DATA_BLOCK "Tor2_RecepturyStacjaMycia"   // DB6
VERSION : 0.1
// stored: AutoNumber true, DBAccessibleFromOPCUA true, InstanceOfName FB_RecepturyStacjaMycia, InstanceOfType FB
"FB_RecepturyStacjaMycia"
BEGIN
   Receptura[0].nazwaReceptury := WSTRING#'Technology';
   Receptura[1].nazwaReceptury := WSTRING#'CIP AGENTS';
   Receptura[2].nazwaReceptury := WSTRING#'CIP Internal';
   Receptura[3].nazwaReceptury := WSTRING#'Technology';
   Receptura[4].nazwaReceptury := WSTRING#'Pasteurizer line';
   Receptura[5].nazwaReceptury := WSTRING#'NF line';
   Receptura[6].nazwaReceptury := WSTRING#'Car line';
   Receptura[7].nazwaReceptury := WSTRING#'Cream line';
   Receptura[8].nazwaReceptury := WSTRING#'Cream line [test]';
   Receptura[9..19].nazwaReceptury := WSTRING#'nazwa receptury';
   Receptura[20].nazwaReceptury := WSTRING#'Cream line';
   Receptura[0].Krok[0..1].nazwaKroku := WSTRING#'Płukanie Zimne';
   Receptura[0].Krok[2].nazwaKroku := WSTRING#'Płukanie Gorące';
   Receptura[0].Krok[3].nazwaKroku := WSTRING#'Ług';
   Receptura[0].Krok[4].nazwaKroku := WSTRING#'Kwas';
   Receptura[0].Krok[5].nazwaKroku := WSTRING#'Płukanie Główne';
   Receptura[0].Krok[6].nazwaKroku := WSTRING#'Dezynfekcja';
   Receptura[1].Krok[0].nazwaKroku := WSTRING#'Płukanie Zimne';
   Receptura[1].Krok[1].nazwaKroku := WSTRING#'Холодне полоскание';
   Receptura[1].Krok[2].nazwaKroku := WSTRING#'Горячее полоскание';
   Receptura[1].Krok[3].nazwaKroku := WSTRING#'ЩЕЛОЧЬ';
   Receptura[1].Krok[4].nazwaKroku := WSTRING#'КИСЛОТА';
   Receptura[1].Krok[5].nazwaKroku := WSTRING#'полоскание';
   Receptura[1].Krok[6].nazwaKroku := WSTRING#'Дезинфекция';
   Receptura[2].Krok[0].nazwaKroku := WSTRING#'Plukanie zimne';
   Receptura[2].Krok[1].nazwaKroku := WSTRING#'Холодне полоскание';
   Receptura[2].Krok[2].nazwaKroku := WSTRING#'Горячее полоскание';
   Receptura[2].Krok[3].nazwaKroku := WSTRING#'ЩЕЛОЧЬ';
   Receptura[2].Krok[4].nazwaKroku := WSTRING#'КИСЛОТА';
   Receptura[2].Krok[5].nazwaKroku := WSTRING#'полоскание';
   Receptura[2].Krok[6].nazwaKroku := WSTRING#'CIP Agents';
   Receptura[3].Krok[0].nazwaKroku := WSTRING#'Płukanie Główne';
   Receptura[3].Krok[1].nazwaKroku := WSTRING#'Холодне полоскание';
   Receptura[3].Krok[2].nazwaKroku := WSTRING#'Горячее полоскание';
   Receptura[3].Krok[3].nazwaKroku := WSTRING#'ЩЕЛОЧЬ';
   Receptura[3].Krok[4].nazwaKroku := WSTRING#'КИСЛОТА';
   Receptura[3].Krok[5].nazwaKroku := WSTRING#'полоскание';
   Receptura[3].Krok[6].nazwaKroku := WSTRING#'Dezynfekcja';
   Receptura[4].Krok[0].nazwaKroku := WSTRING#'Ług';
   Receptura[4].Krok[1].nazwaKroku := WSTRING#'Холодне полоскание';
   Receptura[4].Krok[2].nazwaKroku := WSTRING#'Горячее полоскание';
   Receptura[4].Krok[3].nazwaKroku := WSTRING#'ЩЕЛОЧЬ';
   Receptura[4].Krok[4].nazwaKroku := WSTRING#'КИСЛОТА';
   Receptura[4].Krok[5].nazwaKroku := WSTRING#'полоскание';
   Receptura[4].Krok[6].nazwaKroku := WSTRING#'Dezynfekcja';
   Receptura[5].Krok[0].nazwaKroku := WSTRING#'Kwas';
   Receptura[5].Krok[1].nazwaKroku := WSTRING#'Холодне полоскание';
   Receptura[5].Krok[2].nazwaKroku := WSTRING#'Горячее полоскание';
   Receptura[5].Krok[3].nazwaKroku := WSTRING#'ЩЕЛОЧЬ';
   Receptura[5].Krok[4].nazwaKroku := WSTRING#'КИСЛОТА';
   Receptura[5].Krok[5].nazwaKroku := WSTRING#'полоскание';
   Receptura[5].Krok[6].nazwaKroku := WSTRING#'Dezynfekcja';
   Receptura[6].Krok[0].nazwaKroku := WSTRING#'Ług';
   Receptura[6].Krok[1].nazwaKroku := WSTRING#'Холодне полоскание';
   Receptura[6].Krok[2].nazwaKroku := WSTRING#'Горячее полоскание';
   Receptura[6].Krok[3].nazwaKroku := WSTRING#'ЩЕЛОЧЬ';
   Receptura[6].Krok[4].nazwaKroku := WSTRING#'КИСЛОТА';
   Receptura[6].Krok[5].nazwaKroku := WSTRING#'полоскание';
   Receptura[6].Krok[6].nazwaKroku := WSTRING#'Dezynfekcja';
   Receptura[7].Krok[0].nazwaKroku := WSTRING#'Płukanie Główne';
   Receptura[7].Krok[1].nazwaKroku := WSTRING#'Холодне полоскание';
   Receptura[7].Krok[2].nazwaKroku := WSTRING#'Горячее полоскание';
   Receptura[7].Krok[3].nazwaKroku := WSTRING#'ЩЕЛОЧЬ';
   Receptura[7].Krok[4].nazwaKroku := WSTRING#'КИСЛОТА';
   Receptura[7].Krok[5].nazwaKroku := WSTRING#'полоскание';
   Receptura[7].Krok[6].nazwaKroku := WSTRING#'Dezynfekcja';
   Receptura[8].Krok[0].nazwaKroku := WSTRING#'Płukanie Gorące';
   Receptura[8].Krok[1].nazwaKroku := WSTRING#'Холодне полоскание';
   Receptura[8].Krok[2].nazwaKroku := WSTRING#'Горячее полоскание';
   Receptura[8].Krok[3].nazwaKroku := WSTRING#'ЩЕЛОЧЬ';
   Receptura[8].Krok[4].nazwaKroku := WSTRING#'КИСЛОТА';
   Receptura[8].Krok[5].nazwaKroku := WSTRING#'Płukanie Główne';
   Receptura[8].Krok[6].nazwaKroku := WSTRING#'Dezynfekcja';
   Receptura[9].Krok[0].nazwaKroku := WSTRING#'';
   Receptura[9].Krok[1].nazwaKroku := WSTRING#'Płukanie Zimne';
   Receptura[9].Krok[2].nazwaKroku := WSTRING#'Płukanie Gorące';
   Receptura[9].Krok[3].nazwaKroku := WSTRING#'Ług';
   Receptura[9].Krok[4].nazwaKroku := WSTRING#'Kwas';
   Receptura[9].Krok[5].nazwaKroku := WSTRING#'Płukanie Główne';
   Receptura[9].Krok[6].nazwaKroku := WSTRING#'Dezynfekcja';
   Receptura[10].Krok[0].nazwaKroku := WSTRING#'';
   Receptura[10].Krok[1].nazwaKroku := WSTRING#'Płukanie Zimne';
   Receptura[10].Krok[2].nazwaKroku := WSTRING#'Płukanie Gorące';
   Receptura[10].Krok[3].nazwaKroku := WSTRING#'Ług';
   Receptura[10].Krok[4].nazwaKroku := WSTRING#'Kwas';
   Receptura[10].Krok[5].nazwaKroku := WSTRING#'Płukanie Główne';
   Receptura[10].Krok[6].nazwaKroku := WSTRING#'Dezynfekcja';
   Receptura[11].Krok[0].nazwaKroku := WSTRING#'';
   Receptura[11].Krok[1].nazwaKroku := WSTRING#'Płukanie Zimne';
   Receptura[11].Krok[2].nazwaKroku := WSTRING#'Płukanie Gorące';
   Receptura[11].Krok[3].nazwaKroku := WSTRING#'Ług';
   Receptura[11].Krok[4].nazwaKroku := WSTRING#'Kwas';
   Receptura[11].Krok[5].nazwaKroku := WSTRING#'Płukanie Główne';
   Receptura[11].Krok[6].nazwaKroku := WSTRING#'Dezynfekcja';
   Receptura[12].Krok[0].nazwaKroku := WSTRING#'';
   Receptura[12].Krok[1].nazwaKroku := WSTRING#'Płukanie Zimne';
   Receptura[12].Krok[2].nazwaKroku := WSTRING#'Płukanie Gorące';
   Receptura[12].Krok[3].nazwaKroku := WSTRING#'Ług';
   Receptura[12].Krok[4].nazwaKroku := WSTRING#'Kwas';
   Receptura[12].Krok[5].nazwaKroku := WSTRING#'Płukanie Główne';
   Receptura[12].Krok[6].nazwaKroku := WSTRING#'Dezynfekcja';
   Receptura[13].Krok[0].nazwaKroku := WSTRING#'';
   Receptura[13].Krok[1].nazwaKroku := WSTRING#'Płukanie Zimne';
   Receptura[13].Krok[2].nazwaKroku := WSTRING#'Płukanie Gorące';
   Receptura[13].Krok[3].nazwaKroku := WSTRING#'Ług';
   Receptura[13].Krok[4].nazwaKroku := WSTRING#'Kwas';
   Receptura[13].Krok[5].nazwaKroku := WSTRING#'Płukanie Główne';
   Receptura[13].Krok[6].nazwaKroku := WSTRING#'Dezynfekcja';
   Receptura[14].Krok[0].nazwaKroku := WSTRING#'';
   Receptura[14].Krok[1].nazwaKroku := WSTRING#'Płukanie Zimne';
   Receptura[14].Krok[2].nazwaKroku := WSTRING#'Płukanie Gorące';
   Receptura[14].Krok[3].nazwaKroku := WSTRING#'Ług';
   Receptura[14].Krok[4].nazwaKroku := WSTRING#'Kwas';
   Receptura[14].Krok[5].nazwaKroku := WSTRING#'Płukanie Główne';
   Receptura[14].Krok[6].nazwaKroku := WSTRING#'Dezynfekcja';
   Receptura[15].Krok[0].nazwaKroku := WSTRING#'';
   Receptura[15].Krok[1].nazwaKroku := WSTRING#'Płukanie Zimne';
   Receptura[15].Krok[2].nazwaKroku := WSTRING#'Płukanie Gorące';
   Receptura[15].Krok[3].nazwaKroku := WSTRING#'Ług';
   Receptura[15].Krok[4].nazwaKroku := WSTRING#'Kwas';
   Receptura[15].Krok[5].nazwaKroku := WSTRING#'Płukanie Główne';
   Receptura[15].Krok[6].nazwaKroku := WSTRING#'Dezynfekcja';
   Receptura[16].Krok[0].nazwaKroku := WSTRING#'';
   Receptura[16].Krok[1].nazwaKroku := WSTRING#'Płukanie Zimne';
   Receptura[16].Krok[2].nazwaKroku := WSTRING#'Płukanie Gorące';
   Receptura[16].Krok[3].nazwaKroku := WSTRING#'Ług';
   Receptura[16].Krok[4].nazwaKroku := WSTRING#'Kwas';
   Receptura[16].Krok[5].nazwaKroku := WSTRING#'Płukanie Główne';
   Receptura[16].Krok[6].nazwaKroku := WSTRING#'Dezynfekcja';
   Receptura[17].Krok[0].nazwaKroku := WSTRING#'';
   Receptura[17].Krok[1].nazwaKroku := WSTRING#'Płukanie Zimne';
   Receptura[17].Krok[2].nazwaKroku := WSTRING#'Płukanie Gorące';
   Receptura[17].Krok[3].nazwaKroku := WSTRING#'Ług';
   Receptura[17].Krok[4].nazwaKroku := WSTRING#'Kwas';
   Receptura[17].Krok[5].nazwaKroku := WSTRING#'Płukanie Główne';
   Receptura[17].Krok[6].nazwaKroku := WSTRING#'Dezynfekcja';
   Receptura[18].Krok[0].nazwaKroku := WSTRING#'';
   Receptura[18].Krok[1].nazwaKroku := WSTRING#'Płukanie Zimne';
   Receptura[18].Krok[2].nazwaKroku := WSTRING#'Płukanie Gorące';
   Receptura[18].Krok[3].nazwaKroku := WSTRING#'Ług';
   Receptura[18].Krok[4].nazwaKroku := WSTRING#'Kwas';
   Receptura[18].Krok[5].nazwaKroku := WSTRING#'Płukanie Główne';
   Receptura[18].Krok[6].nazwaKroku := WSTRING#'Dezynfekcja';
   Receptura[19].Krok[0].nazwaKroku := WSTRING#'';
   Receptura[19].Krok[1].nazwaKroku := WSTRING#'Płukanie Zimne';
   Receptura[19].Krok[2].nazwaKroku := WSTRING#'Płukanie Gorące';
   Receptura[19].Krok[3].nazwaKroku := WSTRING#'Ług';
   Receptura[19].Krok[4].nazwaKroku := WSTRING#'Kwas';
   Receptura[19].Krok[5].nazwaKroku := WSTRING#'Płukanie Główne';
   Receptura[19].Krok[6].nazwaKroku := WSTRING#'Dezynfekcja';
   Receptura[20].Krok[0..1].nazwaKroku := WSTRING#'Płukanie Zimne';
   Receptura[20].Krok[2].nazwaKroku := WSTRING#'Płukanie Gorące';
   Receptura[20].Krok[3].nazwaKroku := WSTRING#'Ług';
   Receptura[20].Krok[4].nazwaKroku := WSTRING#'Kwas';
   Receptura[20].Krok[5].nazwaKroku := WSTRING#'Płukanie Główne';
   Receptura[20].Krok[6].nazwaKroku := WSTRING#'Dezynfekcja';
   Receptura[0].Krok[0].PM[0] := 0.0;
   Receptura[0].Krok[0].PM[1] := 1.0;
   Receptura[0].Krok[0].PM[2] := 20.0;
   Receptura[0].Krok[0].PM[3] := 10.0;
   Receptura[0].Krok[0].PM[4] := 120.0;
   Receptura[0].Krok[0].PM[5] := 1.0;
   Receptura[0].Krok[0].PM[6..11] := 0.0;
   Receptura[0].Krok[0].PM[12] := 3.0;
   Receptura[0].Krok[0].PM[13..14] := 0.0;
   Receptura[0].Krok[0].PM[15] := 1.0;
   Receptura[0].Krok[0].PM[16..18] := 0.0;
   Receptura[0].Krok[0].PM[19] := 300.0;
   Receptura[0].Krok[0].PM[20] := 0.0;
   Receptura[0].Krok[0].PM[21] := 1.0;
   Receptura[0].Krok[0].PM[22..23] := 0.0;
   Receptura[0].Krok[0].PM[24] := 2102.0;
   Receptura[0].Krok[0].PM[25..30] := 0.0;
   Receptura[0].Krok[1].PM[0] := 0.0;
   Receptura[0].Krok[1].PM[1] := 1.0;
   Receptura[0].Krok[1].PM[2] := 20.0;
   Receptura[0].Krok[1].PM[3] := 10.0;
   Receptura[0].Krok[1].PM[4] := 120.0;
   Receptura[0].Krok[1].PM[5] := 1.0;
   Receptura[0].Krok[1].PM[6..11] := 0.0;
   Receptura[0].Krok[1].PM[12] := 3.0;
   Receptura[0].Krok[1].PM[13..14] := 0.0;
   Receptura[0].Krok[1].PM[15] := 1.0;
   Receptura[0].Krok[1].PM[16..18] := 0.0;
   Receptura[0].Krok[1].PM[19] := 300.0;
   Receptura[0].Krok[1].PM[20] := 0.0;
   Receptura[0].Krok[1].PM[21] := 1.0;
   Receptura[0].Krok[1].PM[22..23] := 0.0;
   Receptura[0].Krok[1].PM[24] := 2102.0;
   Receptura[0].Krok[1].PM[25..30] := 0.0;
   Receptura[0].Krok[2].PM[0] := 0.0;
   Receptura[0].Krok[2].PM[1] := 1.0;
   Receptura[0].Krok[2].PM[2] := 20.0;
   Receptura[0].Krok[2].PM[3] := 10.0;
   Receptura[0].Krok[2].PM[4] := 120.0;
   Receptura[0].Krok[2].PM[5] := 0.5;
   Receptura[0].Krok[2].PM[6..11] := 0.0;
   Receptura[0].Krok[2].PM[12] := 3.0;
   Receptura[0].Krok[2].PM[13] := 0.0;
   Receptura[0].Krok[2].PM[14] := 30.0;
   Receptura[0].Krok[2].PM[15] := 1.0;
   Receptura[0].Krok[2].PM[16] := 10.0;
   Receptura[0].Krok[2].PM[17..18] := 0.0;
   Receptura[0].Krok[2].PM[19] := 300.0;
   Receptura[0].Krok[2].PM[20] := 0.0;
   Receptura[0].Krok[2].PM[21] := 1.0;
   Receptura[0].Krok[2].PM[22..23] := 0.0;
   Receptura[0].Krok[2].PM[24] := 2102.0;
   Receptura[0].Krok[2].PM[25..30] := 0.0;
   Receptura[0].Krok[3].PM[0] := 0.0;
   Receptura[0].Krok[3].PM[1] := 1.0;
   Receptura[0].Krok[3].PM[2] := 20.0;
   Receptura[0].Krok[3].PM[3] := 10.0;
   Receptura[0].Krok[3].PM[4] := 120.0;
   Receptura[0].Krok[3].PM[5] := 1.0;
   Receptura[0].Krok[3].PM[6] := 900.0;
   Receptura[0].Krok[3].PM[7..9] := 0.0;
   Receptura[0].Krok[3].PM[10] := 40.0;
   Receptura[0].Krok[3].PM[11] := 75.0;
   Receptura[0].Krok[3].PM[12] := 3.0;
   Receptura[0].Krok[3].PM[13] := 70.0;
   Receptura[0].Krok[3].PM[14] := 30.0;
   Receptura[0].Krok[3].PM[15] := 1.0;
   Receptura[0].Krok[3].PM[16] := 10.0;
   Receptura[0].Krok[3].PM[17] := 2.05;
   Receptura[0].Krok[3].PM[18] := 20.0;
   Receptura[0].Krok[3].PM[19] := 300.0;
   Receptura[0].Krok[3].PM[20] := 0.0;
   Receptura[0].Krok[3].PM[21..22] := 1.0;
   Receptura[0].Krok[3].PM[23] := 0.0;
   Receptura[0].Krok[3].PM[24] := 2102.0;
   Receptura[0].Krok[3].PM[25..30] := 0.0;
   Receptura[0].Krok[4].PM[0] := 0.0;
   Receptura[0].Krok[4].PM[1] := 1.0;
   Receptura[0].Krok[4].PM[2] := 20.0;
   Receptura[0].Krok[4].PM[3] := 10.0;
   Receptura[0].Krok[4].PM[4] := 120.0;
   Receptura[0].Krok[4].PM[5] := 0.1;
   Receptura[0].Krok[4].PM[6] := 300.0;
   Receptura[0].Krok[4].PM[7..9] := 0.0;
   Receptura[0].Krok[4].PM[10] := 30.0;
   Receptura[0].Krok[4].PM[11] := 50.0;
   Receptura[0].Krok[4].PM[12] := 3.0;
   Receptura[0].Krok[4].PM[13] := 55.0;
   Receptura[0].Krok[4].PM[14] := 0.0;
   Receptura[0].Krok[4].PM[15] := 1.0;
   Receptura[0].Krok[4].PM[16] := 10.0;
   Receptura[0].Krok[4].PM[17] := 1.75;
   Receptura[0].Krok[4].PM[18] := 20.0;
   Receptura[0].Krok[4].PM[19] := 300.0;
   Receptura[0].Krok[4].PM[20] := 0.0;
   Receptura[0].Krok[4].PM[21..22] := 1.0;
   Receptura[0].Krok[4].PM[23] := 0.0;
   Receptura[0].Krok[4].PM[24] := 2102.0;
   Receptura[0].Krok[4].PM[25..30] := 0.0;
   Receptura[0].Krok[5].PM[0] := 0.0;
   Receptura[0].Krok[5].PM[1] := 1.0;
   Receptura[0].Krok[5].PM[2] := 20.0;
   Receptura[0].Krok[5].PM[3] := 10.0;
   Receptura[0].Krok[5].PM[4] := 120.0;
   Receptura[0].Krok[5].PM[5] := 1.25;
   Receptura[0].Krok[5].PM[6..11] := 0.0;
   Receptura[0].Krok[5].PM[12] := 3.0;
   Receptura[0].Krok[5].PM[13..14] := 0.0;
   Receptura[0].Krok[5].PM[15] := 1.0;
   Receptura[0].Krok[5].PM[16] := 5.0;
   Receptura[0].Krok[5].PM[17..18] := 0.0;
   Receptura[0].Krok[5].PM[19] := 300.0;
   Receptura[0].Krok[5].PM[20] := 0.0;
   Receptura[0].Krok[5].PM[21] := 1.0;
   Receptura[0].Krok[5].PM[22..23] := 0.0;
   Receptura[0].Krok[5].PM[24] := 2102.0;
   Receptura[0].Krok[5].PM[25..30] := 0.0;
   Receptura[0].Krok[6].PM[0..30] := 0.0;
   Receptura[1].Krok[0].PM[0..1] := 0.0;
   Receptura[1].Krok[0].PM[2] := 25.0;
   Receptura[1].Krok[0].PM[3] := 10.0;
   Receptura[1].Krok[0].PM[4] := 120.0;
   Receptura[1].Krok[0].PM[5] := 1.0;
   Receptura[1].Krok[0].PM[6..11] := 0.0;
   Receptura[1].Krok[0].PM[12] := 3.0;
   Receptura[1].Krok[0].PM[13..14] := 0.0;
   Receptura[1].Krok[0].PM[15] := 1.0;
   Receptura[1].Krok[0].PM[16..18] := 0.0;
   Receptura[1].Krok[0].PM[19] := 300.0;
   Receptura[1].Krok[0].PM[20..22] := 0.0;
   Receptura[1].Krok[0].PM[23] := 1.0;
   Receptura[1].Krok[0].PM[24] := 9401.0;
   Receptura[1].Krok[0].PM[25..30] := 0.0;
   Receptura[1].Krok[1].PM[0..1] := 0.0;
   Receptura[1].Krok[1].PM[2] := 25.0;
   Receptura[1].Krok[1].PM[3] := 10.0;
   Receptura[1].Krok[1].PM[4] := 120.0;
   Receptura[1].Krok[1].PM[5] := 1.0;
   Receptura[1].Krok[1].PM[6..11] := 0.0;
   Receptura[1].Krok[1].PM[12] := 3.0;
   Receptura[1].Krok[1].PM[13..14] := 0.0;
   Receptura[1].Krok[1].PM[15] := 1.0;
   Receptura[1].Krok[1].PM[16..18] := 0.0;
   Receptura[1].Krok[1].PM[19] := 300.0;
   Receptura[1].Krok[1].PM[20..22] := 0.0;
   Receptura[1].Krok[1].PM[23] := 1.0;
   Receptura[1].Krok[1].PM[24] := 9401.0;
   Receptura[1].Krok[1].PM[25..30] := 0.0;
   Receptura[1].Krok[2].PM[0..1] := 0.0;
   Receptura[1].Krok[2].PM[2] := 25.0;
   Receptura[1].Krok[2].PM[3] := 10.0;
   Receptura[1].Krok[2].PM[4] := 120.0;
   Receptura[1].Krok[2].PM[5] := 0.5;
   Receptura[1].Krok[2].PM[6..11] := 0.0;
   Receptura[1].Krok[2].PM[12] := 3.0;
   Receptura[1].Krok[2].PM[13] := 0.0;
   Receptura[1].Krok[2].PM[14] := 30.0;
   Receptura[1].Krok[2].PM[15] := 1.0;
   Receptura[1].Krok[2].PM[16] := 10.0;
   Receptura[1].Krok[2].PM[17..18] := 0.0;
   Receptura[1].Krok[2].PM[19] := 300.0;
   Receptura[1].Krok[2].PM[20..22] := 0.0;
   Receptura[1].Krok[2].PM[23] := 1.0;
   Receptura[1].Krok[2].PM[24] := 9401.0;
   Receptura[1].Krok[2].PM[25..30] := 0.0;
   Receptura[1].Krok[3].PM[0..1] := 0.0;
   Receptura[1].Krok[3].PM[2] := 25.0;
   Receptura[1].Krok[3].PM[3] := 10.0;
   Receptura[1].Krok[3].PM[4] := 120.0;
   Receptura[1].Krok[3].PM[5] := 1.0;
   Receptura[1].Krok[3].PM[6] := 900.0;
   Receptura[1].Krok[3].PM[7..9] := 0.0;
   Receptura[1].Krok[3].PM[10] := 60.0;
   Receptura[1].Krok[3].PM[11] := 75.0;
   Receptura[1].Krok[3].PM[12] := 3.0;
   Receptura[1].Krok[3].PM[13] := 70.0;
   Receptura[1].Krok[3].PM[14] := 30.0;
   Receptura[1].Krok[3].PM[15] := 1.0;
   Receptura[1].Krok[3].PM[16] := 10.0;
   Receptura[1].Krok[3].PM[17] := 2.05;
   Receptura[1].Krok[3].PM[18] := 20.0;
   Receptura[1].Krok[3].PM[19] := 300.0;
   Receptura[1].Krok[3].PM[20..21] := 0.0;
   Receptura[1].Krok[3].PM[22] := 1.0;
   Receptura[1].Krok[3].PM[23] := 0.0;
   Receptura[1].Krok[3].PM[24] := 9401.0;
   Receptura[1].Krok[3].PM[25..30] := 0.0;
   Receptura[1].Krok[4].PM[0] := 0.0;
   Receptura[1].Krok[4].PM[1] := 1.0;
   Receptura[1].Krok[4].PM[2] := 22.0;
   Receptura[1].Krok[4].PM[3] := 10.0;
   Receptura[1].Krok[4].PM[4] := 120.0;
   Receptura[1].Krok[4].PM[5] := 0.1;
   Receptura[1].Krok[4].PM[6] := 300.0;
   Receptura[1].Krok[4].PM[7..9] := 0.0;
   Receptura[1].Krok[4].PM[10] := 35.0;
   Receptura[1].Krok[4].PM[11] := 50.0;
   Receptura[1].Krok[4].PM[12] := 3.0;
   Receptura[1].Krok[4].PM[13] := 60.0;
   Receptura[1].Krok[4].PM[14] := 0.0;
   Receptura[1].Krok[4].PM[15] := 1.0;
   Receptura[1].Krok[4].PM[16] := 10.0;
   Receptura[1].Krok[4].PM[17] := 1.75;
   Receptura[1].Krok[4].PM[18] := 20.0;
   Receptura[1].Krok[4].PM[19] := 300.0;
   Receptura[1].Krok[4].PM[20..21] := 0.0;
   Receptura[1].Krok[4].PM[22..23] := 1.0;
   Receptura[1].Krok[4].PM[24] := 9401.0;
   Receptura[1].Krok[4].PM[25..30] := 0.0;
   Receptura[1].Krok[5].PM[0] := 0.0;
   Receptura[1].Krok[5].PM[1] := 1.0;
   Receptura[1].Krok[5].PM[2] := 25.0;
   Receptura[1].Krok[5].PM[3] := 10.0;
   Receptura[1].Krok[5].PM[4] := 120.0;
   Receptura[1].Krok[5].PM[5] := 1.5;
   Receptura[1].Krok[5].PM[6..11] := 0.0;
   Receptura[1].Krok[5].PM[12] := 3.0;
   Receptura[1].Krok[5].PM[13..14] := 0.0;
   Receptura[1].Krok[5].PM[15] := 1.0;
   Receptura[1].Krok[5].PM[16..18] := 0.0;
   Receptura[1].Krok[5].PM[19] := 300.0;
   Receptura[1].Krok[5].PM[20..22] := 0.0;
   Receptura[1].Krok[5].PM[23] := 1.0;
   Receptura[1].Krok[5].PM[24] := 9401.0;
   Receptura[1].Krok[5].PM[25..30] := 0.0;
   Receptura[1].Krok[6].PM[0..30] := 0.0;
   Receptura[2].Krok[0].PM[0] := 0.0;
   Receptura[2].Krok[0].PM[1] := 1.0;
   Receptura[2].Krok[0].PM[2] := 20.0;
   Receptura[2].Krok[0].PM[3] := 10.0;
   Receptura[2].Krok[0].PM[4] := 30.0;
   Receptura[2].Krok[0].PM[5] := 1.0;
   Receptura[2].Krok[0].PM[6] := 0.0;
   Receptura[2].Krok[0].PM[7] := 5.0;
   Receptura[2].Krok[0].PM[8] := 0.0;
   Receptura[2].Krok[0].PM[9] := 5.0;
   Receptura[2].Krok[0].PM[10..11] := 0.0;
   Receptura[2].Krok[0].PM[12] := 3.0;
   Receptura[2].Krok[0].PM[13..14] := 0.0;
   Receptura[2].Krok[0].PM[15] := 1.0;
   Receptura[2].Krok[0].PM[16] := 5.0;
   Receptura[2].Krok[0].PM[17..18] := 0.0;
   Receptura[2].Krok[0].PM[19] := 300.0;
   Receptura[2].Krok[0].PM[20..22] := 0.0;
   Receptura[2].Krok[0].PM[23] := 1.0;
   Receptura[2].Krok[0].PM[24..30] := 0.0;
   Receptura[2].Krok[1].PM[0] := 0.0;
   Receptura[2].Krok[1].PM[1] := 1.0;
   Receptura[2].Krok[1].PM[2] := 20.0;
   Receptura[2].Krok[1].PM[3] := 10.0;
   Receptura[2].Krok[1].PM[4] := 30.0;
   Receptura[2].Krok[1].PM[5] := 1.0;
   Receptura[2].Krok[1].PM[6] := 0.0;
   Receptura[2].Krok[1].PM[7] := 5.0;
   Receptura[2].Krok[1].PM[8] := 0.0;
   Receptura[2].Krok[1].PM[9] := 5.0;
   Receptura[2].Krok[1].PM[10..11] := 0.0;
   Receptura[2].Krok[1].PM[12] := 3.0;
   Receptura[2].Krok[1].PM[13..14] := 0.0;
   Receptura[2].Krok[1].PM[15] := 1.0;
   Receptura[2].Krok[1].PM[16] := 5.0;
   Receptura[2].Krok[1].PM[17..18] := 0.0;
   Receptura[2].Krok[1].PM[19] := 300.0;
   Receptura[2].Krok[1].PM[20..22] := 0.0;
   Receptura[2].Krok[1].PM[23] := 1.0;
   Receptura[2].Krok[1].PM[24..30] := 0.0;
   Receptura[2].Krok[2].PM[0] := 0.0;
   Receptura[2].Krok[2].PM[1] := 1.0;
   Receptura[2].Krok[2].PM[2] := 20.0;
   Receptura[2].Krok[2].PM[3] := 10.0;
   Receptura[2].Krok[2].PM[4] := 30.0;
   Receptura[2].Krok[2].PM[5] := 1.0;
   Receptura[2].Krok[2].PM[6] := 0.0;
   Receptura[2].Krok[2].PM[7] := 5.0;
   Receptura[2].Krok[2].PM[8] := 0.0;
   Receptura[2].Krok[2].PM[9] := 5.0;
   Receptura[2].Krok[2].PM[10..11] := 0.0;
   Receptura[2].Krok[2].PM[12] := 3.0;
   Receptura[2].Krok[2].PM[13] := 0.0;
   Receptura[2].Krok[2].PM[14] := 30.0;
   Receptura[2].Krok[2].PM[15] := 1.0;
   Receptura[2].Krok[2].PM[16] := 5.0;
   Receptura[2].Krok[2].PM[17..18] := 0.0;
   Receptura[2].Krok[2].PM[19] := 300.0;
   Receptura[2].Krok[2].PM[20..22] := 0.0;
   Receptura[2].Krok[2].PM[23] := 1.0;
   Receptura[2].Krok[2].PM[24..30] := 0.0;
   Receptura[2].Krok[3].PM[0] := 0.0;
   Receptura[2].Krok[3].PM[1] := 1.0;
   Receptura[2].Krok[3].PM[2] := 20.0;
   Receptura[2].Krok[3].PM[3] := 10.0;
   Receptura[2].Krok[3].PM[4] := 30.0;
   Receptura[2].Krok[3].PM[5] := 2.0;
   Receptura[2].Krok[3].PM[6] := 600.0;
   Receptura[2].Krok[3].PM[7] := 5.0;
   Receptura[2].Krok[3].PM[8] := 0.0;
   Receptura[2].Krok[3].PM[9] := 5.0;
   Receptura[2].Krok[3].PM[10] := 60.0;
   Receptura[2].Krok[3].PM[11] := 75.0;
   Receptura[2].Krok[3].PM[12] := 3.0;
   Receptura[2].Krok[3].PM[13] := 70.0;
   Receptura[2].Krok[3].PM[14] := 30.0;
   Receptura[2].Krok[3].PM[15] := 1.0;
   Receptura[2].Krok[3].PM[16] := 5.0;
   Receptura[2].Krok[3].PM[17] := 2.05;
   Receptura[2].Krok[3].PM[18] := 20.0;
   Receptura[2].Krok[3].PM[19] := 300.0;
   Receptura[2].Krok[3].PM[20..21] := 0.0;
   Receptura[2].Krok[3].PM[22..23] := 1.0;
   Receptura[2].Krok[3].PM[24..30] := 0.0;
   Receptura[2].Krok[4].PM[0] := 0.0;
   Receptura[2].Krok[4].PM[1] := 1.0;
   Receptura[2].Krok[4].PM[2] := 20.0;
   Receptura[2].Krok[4].PM[3] := 10.0;
   Receptura[2].Krok[4].PM[4] := 30.0;
   Receptura[2].Krok[4].PM[5] := 1.0;
   Receptura[2].Krok[4].PM[6] := 300.0;
   Receptura[2].Krok[4].PM[7] := 5.0;
   Receptura[2].Krok[4].PM[8] := 0.0;
   Receptura[2].Krok[4].PM[9] := 5.0;
   Receptura[2].Krok[4].PM[10] := 35.0;
   Receptura[2].Krok[4].PM[11] := 50.0;
   Receptura[2].Krok[4].PM[12] := 3.0;
   Receptura[2].Krok[4].PM[13] := 60.0;
   Receptura[2].Krok[4].PM[14] := 30.0;
   Receptura[2].Krok[4].PM[15] := 1.0;
   Receptura[2].Krok[4].PM[16] := 5.0;
   Receptura[2].Krok[4].PM[17] := 1.75;
   Receptura[2].Krok[4].PM[18] := 20.0;
   Receptura[2].Krok[4].PM[19] := 300.0;
   Receptura[2].Krok[4].PM[20..21] := 0.0;
   Receptura[2].Krok[4].PM[22..23] := 1.0;
   Receptura[2].Krok[4].PM[24..30] := 0.0;
   Receptura[2].Krok[5].PM[0] := 0.0;
   Receptura[2].Krok[5].PM[1] := 1.0;
   Receptura[2].Krok[5].PM[2] := 20.0;
   Receptura[2].Krok[5].PM[3] := 10.0;
   Receptura[2].Krok[5].PM[4] := 30.0;
   Receptura[2].Krok[5].PM[5] := 2.0;
   Receptura[2].Krok[5].PM[6] := 0.0;
   Receptura[2].Krok[5].PM[7] := 5.0;
   Receptura[2].Krok[5].PM[8] := 0.0;
   Receptura[2].Krok[5].PM[9] := 5.0;
   Receptura[2].Krok[5].PM[10..11] := 0.0;
   Receptura[2].Krok[5].PM[12] := 3.0;
   Receptura[2].Krok[5].PM[13..14] := 0.0;
   Receptura[2].Krok[5].PM[15] := 1.0;
   Receptura[2].Krok[5].PM[16..18] := 0.0;
   Receptura[2].Krok[5].PM[19] := 300.0;
   Receptura[2].Krok[5].PM[20..22] := 0.0;
   Receptura[2].Krok[5].PM[23] := 1.0;
   Receptura[2].Krok[5].PM[24..30] := 0.0;
   Receptura[2].Krok[6].PM[0..30] := 0.0;
   Receptura[3].Krok[0].PM[0] := 0.0;
   Receptura[3].Krok[0].PM[1] := 1.0;
   Receptura[3].Krok[0].PM[2] := 20.0;
   Receptura[3].Krok[0].PM[3] := 10.0;
   Receptura[3].Krok[0].PM[4] := 120.0;
   Receptura[3].Krok[0].PM[5] := 1.25;
   Receptura[3].Krok[0].PM[6..11] := 0.0;
   Receptura[3].Krok[0].PM[12] := 3.0;
   Receptura[3].Krok[0].PM[13..14] := 0.0;
   Receptura[3].Krok[0].PM[15] := 1.0;
   Receptura[3].Krok[0].PM[16] := 5.0;
   Receptura[3].Krok[0].PM[17..18] := 0.0;
   Receptura[3].Krok[0].PM[19] := 300.0;
   Receptura[3].Krok[0].PM[20] := 0.0;
   Receptura[3].Krok[0].PM[21] := 1.0;
   Receptura[3].Krok[0].PM[22..23] := 0.0;
   Receptura[3].Krok[0].PM[24] := 2102.0;
   Receptura[3].Krok[0].PM[25..30] := 0.0;
   Receptura[3].Krok[1].PM[0] := 0.0;
   Receptura[3].Krok[1].PM[1] := 1.0;
   Receptura[3].Krok[1].PM[2] := 20.0;
   Receptura[3].Krok[1].PM[3] := 10.0;
   Receptura[3].Krok[1].PM[4] := 120.0;
   Receptura[3].Krok[1].PM[5] := 1.0;
   Receptura[3].Krok[1].PM[6..11] := 0.0;
   Receptura[3].Krok[1].PM[12] := 3.0;
   Receptura[3].Krok[1].PM[13..14] := 0.0;
   Receptura[3].Krok[1].PM[15] := 1.0;
   Receptura[3].Krok[1].PM[16..18] := 0.0;
   Receptura[3].Krok[1].PM[19] := 300.0;
   Receptura[3].Krok[1].PM[20] := 0.0;
   Receptura[3].Krok[1].PM[21] := 1.0;
   Receptura[3].Krok[1].PM[22..23] := 0.0;
   Receptura[3].Krok[1].PM[24] := 2102.0;
   Receptura[3].Krok[1].PM[25..30] := 0.0;
   Receptura[3].Krok[2].PM[0] := 0.0;
   Receptura[3].Krok[2].PM[1] := 1.0;
   Receptura[3].Krok[2].PM[2] := 20.0;
   Receptura[3].Krok[2].PM[3] := 10.0;
   Receptura[3].Krok[2].PM[4] := 120.0;
   Receptura[3].Krok[2].PM[5] := 0.5;
   Receptura[3].Krok[2].PM[6..11] := 0.0;
   Receptura[3].Krok[2].PM[12] := 3.0;
   Receptura[3].Krok[2].PM[13] := 0.0;
   Receptura[3].Krok[2].PM[14] := 30.0;
   Receptura[3].Krok[2].PM[15] := 1.0;
   Receptura[3].Krok[2].PM[16] := 10.0;
   Receptura[3].Krok[2].PM[17..18] := 0.0;
   Receptura[3].Krok[2].PM[19] := 300.0;
   Receptura[3].Krok[2].PM[20] := 0.0;
   Receptura[3].Krok[2].PM[21] := 1.0;
   Receptura[3].Krok[2].PM[22..23] := 0.0;
   Receptura[3].Krok[2].PM[24] := 2102.0;
   Receptura[3].Krok[2].PM[25..30] := 0.0;
   Receptura[3].Krok[3].PM[0] := 0.0;
   Receptura[3].Krok[3].PM[1] := 1.0;
   Receptura[3].Krok[3].PM[2] := 20.0;
   Receptura[3].Krok[3].PM[3] := 10.0;
   Receptura[3].Krok[3].PM[4] := 120.0;
   Receptura[3].Krok[3].PM[5] := 1.0;
   Receptura[3].Krok[3].PM[6] := 900.0;
   Receptura[3].Krok[3].PM[7..9] := 0.0;
   Receptura[3].Krok[3].PM[10] := 40.0;
   Receptura[3].Krok[3].PM[11] := 75.0;
   Receptura[3].Krok[3].PM[12] := 3.0;
   Receptura[3].Krok[3].PM[13] := 70.0;
   Receptura[3].Krok[3].PM[14] := 30.0;
   Receptura[3].Krok[3].PM[15] := 1.0;
   Receptura[3].Krok[3].PM[16] := 10.0;
   Receptura[3].Krok[3].PM[17] := 2.05;
   Receptura[3].Krok[3].PM[18] := 20.0;
   Receptura[3].Krok[3].PM[19] := 300.0;
   Receptura[3].Krok[3].PM[20] := 0.0;
   Receptura[3].Krok[3].PM[21..22] := 1.0;
   Receptura[3].Krok[3].PM[23] := 0.0;
   Receptura[3].Krok[3].PM[24] := 2102.0;
   Receptura[3].Krok[3].PM[25..30] := 0.0;
   Receptura[3].Krok[4].PM[0] := 0.0;
   Receptura[3].Krok[4].PM[1] := 1.0;
   Receptura[3].Krok[4].PM[2] := 20.0;
   Receptura[3].Krok[4].PM[3] := 10.0;
   Receptura[3].Krok[4].PM[4] := 120.0;
   Receptura[3].Krok[4].PM[5] := 0.1;
   Receptura[3].Krok[4].PM[6] := 300.0;
   Receptura[3].Krok[4].PM[7..9] := 0.0;
   Receptura[3].Krok[4].PM[10] := 30.0;
   Receptura[3].Krok[4].PM[11] := 50.0;
   Receptura[3].Krok[4].PM[12] := 3.0;
   Receptura[3].Krok[4].PM[13] := 55.0;
   Receptura[3].Krok[4].PM[14] := 0.0;
   Receptura[3].Krok[4].PM[15] := 1.0;
   Receptura[3].Krok[4].PM[16] := 10.0;
   Receptura[3].Krok[4].PM[17] := 1.75;
   Receptura[3].Krok[4].PM[18] := 20.0;
   Receptura[3].Krok[4].PM[19] := 300.0;
   Receptura[3].Krok[4].PM[20] := 0.0;
   Receptura[3].Krok[4].PM[21..22] := 1.0;
   Receptura[3].Krok[4].PM[23] := 0.0;
   Receptura[3].Krok[4].PM[24] := 2102.0;
   Receptura[3].Krok[4].PM[25..30] := 0.0;
   Receptura[3].Krok[5].PM[0] := 0.0;
   Receptura[3].Krok[5].PM[1] := 1.0;
   Receptura[3].Krok[5].PM[2] := 20.0;
   Receptura[3].Krok[5].PM[3] := 10.0;
   Receptura[3].Krok[5].PM[4] := 120.0;
   Receptura[3].Krok[5].PM[5] := 1.25;
   Receptura[3].Krok[5].PM[6..11] := 0.0;
   Receptura[3].Krok[5].PM[12] := 3.0;
   Receptura[3].Krok[5].PM[13..14] := 0.0;
   Receptura[3].Krok[5].PM[15] := 1.0;
   Receptura[3].Krok[5].PM[16] := 5.0;
   Receptura[3].Krok[5].PM[17..18] := 0.0;
   Receptura[3].Krok[5].PM[19] := 300.0;
   Receptura[3].Krok[5].PM[20] := 0.0;
   Receptura[3].Krok[5].PM[21] := 1.0;
   Receptura[3].Krok[5].PM[22..23] := 0.0;
   Receptura[3].Krok[5].PM[24] := 2102.0;
   Receptura[3].Krok[5].PM[25..30] := 0.0;
   Receptura[3].Krok[6].PM[0..30] := 0.0;
   Receptura[4].Krok[0].PM[0] := 0.0;
   Receptura[4].Krok[0].PM[1] := 1.0;
   Receptura[4].Krok[0].PM[2] := 20.0;
   Receptura[4].Krok[0].PM[3] := 10.0;
   Receptura[4].Krok[0].PM[4] := 120.0;
   Receptura[4].Krok[0].PM[5] := 1.0;
   Receptura[4].Krok[0].PM[6] := 600.0;
   Receptura[4].Krok[0].PM[7..9] := 0.0;
   Receptura[4].Krok[0].PM[10] := 40.0;
   Receptura[4].Krok[0].PM[11] := 75.0;
   Receptura[4].Krok[0].PM[12] := 3.0;
   Receptura[4].Krok[0].PM[13] := 70.0;
   Receptura[4].Krok[0].PM[14] := 30.0;
   Receptura[4].Krok[0].PM[15] := 1.0;
   Receptura[4].Krok[0].PM[16] := 10.0;
   Receptura[4].Krok[0].PM[17] := 2.05;
   Receptura[4].Krok[0].PM[18] := 20.0;
   Receptura[4].Krok[0].PM[19] := 300.0;
   Receptura[4].Krok[0].PM[20] := 0.0;
   Receptura[4].Krok[0].PM[21..22] := 1.0;
   Receptura[4].Krok[0].PM[23] := 0.0;
   Receptura[4].Krok[0].PM[24] := 2101.0;
   Receptura[4].Krok[0].PM[25..30] := 0.0;
   Receptura[4].Krok[1].PM[0] := 0.0;
   Receptura[4].Krok[1].PM[1] := 1.0;
   Receptura[4].Krok[1].PM[2] := 20.0;
   Receptura[4].Krok[1].PM[3] := 10.0;
   Receptura[4].Krok[1].PM[4] := 120.0;
   Receptura[4].Krok[1].PM[5] := 0.8;
   Receptura[4].Krok[1].PM[6..11] := 0.0;
   Receptura[4].Krok[1].PM[12] := 3.0;
   Receptura[4].Krok[1].PM[13..14] := 0.0;
   Receptura[4].Krok[1].PM[15] := 1.0;
   Receptura[4].Krok[1].PM[16..20] := 0.0;
   Receptura[4].Krok[1].PM[21] := 1.0;
   Receptura[4].Krok[1].PM[22..23] := 0.0;
   Receptura[4].Krok[1].PM[24] := 2101.0;
   Receptura[4].Krok[1].PM[25..30] := 0.0;
   Receptura[4].Krok[2].PM[0] := 0.0;
   Receptura[4].Krok[2].PM[1] := 1.0;
   Receptura[4].Krok[2].PM[2] := 20.0;
   Receptura[4].Krok[2].PM[3] := 10.0;
   Receptura[4].Krok[2].PM[4] := 120.0;
   Receptura[4].Krok[2].PM[5] := 0.5;
   Receptura[4].Krok[2].PM[6..11] := 0.0;
   Receptura[4].Krok[2].PM[12] := 3.0;
   Receptura[4].Krok[2].PM[13] := 0.0;
   Receptura[4].Krok[2].PM[14] := 30.0;
   Receptura[4].Krok[2].PM[15] := 1.0;
   Receptura[4].Krok[2].PM[16] := 10.0;
   Receptura[4].Krok[2].PM[17..18] := 0.0;
   Receptura[4].Krok[2].PM[19] := 300.0;
   Receptura[4].Krok[2].PM[20] := 0.0;
   Receptura[4].Krok[2].PM[21] := 1.0;
   Receptura[4].Krok[2].PM[22..23] := 0.0;
   Receptura[4].Krok[2].PM[24] := 2101.0;
   Receptura[4].Krok[2].PM[25..30] := 0.0;
   Receptura[4].Krok[3].PM[0] := 0.0;
   Receptura[4].Krok[3].PM[1] := 1.0;
   Receptura[4].Krok[3].PM[2] := 20.0;
   Receptura[4].Krok[3].PM[3] := 10.0;
   Receptura[4].Krok[3].PM[4] := 120.0;
   Receptura[4].Krok[3].PM[5] := 1.0;
   Receptura[4].Krok[3].PM[6] := 600.0;
   Receptura[4].Krok[3].PM[7..9] := 0.0;
   Receptura[4].Krok[3].PM[10] := 40.0;
   Receptura[4].Krok[3].PM[11] := 75.0;
   Receptura[4].Krok[3].PM[12] := 3.0;
   Receptura[4].Krok[3].PM[13] := 70.0;
   Receptura[4].Krok[3].PM[14] := 30.0;
   Receptura[4].Krok[3].PM[15] := 1.0;
   Receptura[4].Krok[3].PM[16] := 10.0;
   Receptura[4].Krok[3].PM[17] := 2.05;
   Receptura[4].Krok[3].PM[18] := 20.0;
   Receptura[4].Krok[3].PM[19] := 300.0;
   Receptura[4].Krok[3].PM[20] := 0.0;
   Receptura[4].Krok[3].PM[21..22] := 1.0;
   Receptura[4].Krok[3].PM[23] := 0.0;
   Receptura[4].Krok[3].PM[24] := 2101.0;
   Receptura[4].Krok[3].PM[25..30] := 0.0;
   Receptura[4].Krok[4].PM[0] := 0.0;
   Receptura[4].Krok[4].PM[1] := 1.0;
   Receptura[4].Krok[4].PM[2] := 20.0;
   Receptura[4].Krok[4].PM[3] := 10.0;
   Receptura[4].Krok[4].PM[4] := 120.0;
   Receptura[4].Krok[4].PM[5] := 0.1;
   Receptura[4].Krok[4].PM[6] := 300.0;
   Receptura[4].Krok[4].PM[7..9] := 0.0;
   Receptura[4].Krok[4].PM[10] := 30.0;
   Receptura[4].Krok[4].PM[11] := 50.0;
   Receptura[4].Krok[4].PM[12] := 3.0;
   Receptura[4].Krok[4].PM[13] := 55.0;
   Receptura[4].Krok[4].PM[14] := 0.0;
   Receptura[4].Krok[4].PM[15] := 1.0;
   Receptura[4].Krok[4].PM[16] := 10.0;
   Receptura[4].Krok[4].PM[17] := 1.75;
   Receptura[4].Krok[4].PM[18] := 20.0;
   Receptura[4].Krok[4].PM[19] := 300.0;
   Receptura[4].Krok[4].PM[20] := 0.0;
   Receptura[4].Krok[4].PM[21..22] := 1.0;
   Receptura[4].Krok[4].PM[23] := 0.0;
   Receptura[4].Krok[4].PM[24] := 2101.0;
   Receptura[4].Krok[4].PM[25..30] := 0.0;
   Receptura[4].Krok[5].PM[0] := 0.0;
   Receptura[4].Krok[5].PM[1] := 1.0;
   Receptura[4].Krok[5].PM[2] := 20.0;
   Receptura[4].Krok[5].PM[3] := 10.0;
   Receptura[4].Krok[5].PM[4] := 120.0;
   Receptura[4].Krok[5].PM[5] := 1.5;
   Receptura[4].Krok[5].PM[6..11] := 0.0;
   Receptura[4].Krok[5].PM[12] := 3.0;
   Receptura[4].Krok[5].PM[13..14] := 0.0;
   Receptura[4].Krok[5].PM[15] := 1.0;
   Receptura[4].Krok[5].PM[16..18] := 0.0;
   Receptura[4].Krok[5].PM[19] := 300.0;
   Receptura[4].Krok[5].PM[20] := 0.0;
   Receptura[4].Krok[5].PM[21] := 1.0;
   Receptura[4].Krok[5].PM[22..23] := 0.0;
   Receptura[4].Krok[5].PM[24] := 2101.0;
   Receptura[4].Krok[5].PM[25..30] := 0.0;
   Receptura[4].Krok[6].PM[0..30] := 0.0;
   Receptura[5].Krok[0].PM[0] := 0.0;
   Receptura[5].Krok[0].PM[1] := 1.0;
   Receptura[5].Krok[0].PM[2] := 15.0;
   Receptura[5].Krok[0].PM[3] := 10.0;
   Receptura[5].Krok[0].PM[4] := 60.0;
   Receptura[5].Krok[0].PM[5] := 0.1;
   Receptura[5].Krok[0].PM[6] := 300.0;
   Receptura[5].Krok[0].PM[7..9] := 0.0;
   Receptura[5].Krok[0].PM[10] := 30.0;
   Receptura[5].Krok[0].PM[11] := 50.0;
   Receptura[5].Krok[0].PM[12] := 3.0;
   Receptura[5].Krok[0].PM[13] := 60.0;
   Receptura[5].Krok[0].PM[14] := 0.0;
   Receptura[5].Krok[0].PM[15] := 1.0;
   Receptura[5].Krok[0].PM[16] := 10.0;
   Receptura[5].Krok[0].PM[17] := 1.75;
   Receptura[5].Krok[0].PM[18] := 20.0;
   Receptura[5].Krok[0].PM[19] := 300.0;
   Receptura[5].Krok[0].PM[20] := 0.0;
   Receptura[5].Krok[0].PM[21..22] := 1.0;
   Receptura[5].Krok[0].PM[23] := 0.0;
   Receptura[5].Krok[0].PM[24] := 3101.0;
   Receptura[5].Krok[0].PM[25..30] := 0.0;
   Receptura[5].Krok[1].PM[0] := 0.0;
   Receptura[5].Krok[1].PM[1] := 1.0;
   Receptura[5].Krok[1].PM[2] := 15.0;
   Receptura[5].Krok[1].PM[3] := 10.0;
   Receptura[5].Krok[1].PM[4] := 60.0;
   Receptura[5].Krok[1].PM[5] := 1.0;
   Receptura[5].Krok[1].PM[6..11] := 0.0;
   Receptura[5].Krok[1].PM[12] := 3.0;
   Receptura[5].Krok[1].PM[13..14] := 0.0;
   Receptura[5].Krok[1].PM[15] := 1.0;
   Receptura[5].Krok[1].PM[16..18] := 0.0;
   Receptura[5].Krok[1].PM[19] := 300.0;
   Receptura[5].Krok[1].PM[20] := 0.0;
   Receptura[5].Krok[1].PM[21] := 1.0;
   Receptura[5].Krok[1].PM[22..23] := 0.0;
   Receptura[5].Krok[1].PM[24] := 3101.0;
   Receptura[5].Krok[1].PM[25..30] := 0.0;
   Receptura[5].Krok[2].PM[0] := 0.0;
   Receptura[5].Krok[2].PM[1] := 1.0;
   Receptura[5].Krok[2].PM[2] := 15.0;
   Receptura[5].Krok[2].PM[3] := 10.0;
   Receptura[5].Krok[2].PM[4] := 60.0;
   Receptura[5].Krok[2].PM[5] := 0.5;
   Receptura[5].Krok[2].PM[6..11] := 0.0;
   Receptura[5].Krok[2].PM[12] := 3.0;
   Receptura[5].Krok[2].PM[13] := 0.0;
   Receptura[5].Krok[2].PM[14] := 30.0;
   Receptura[5].Krok[2].PM[15] := 1.0;
   Receptura[5].Krok[2].PM[16] := 10.0;
   Receptura[5].Krok[2].PM[17..18] := 0.0;
   Receptura[5].Krok[2].PM[19] := 300.0;
   Receptura[5].Krok[2].PM[20] := 0.0;
   Receptura[5].Krok[2].PM[21] := 1.0;
   Receptura[5].Krok[2].PM[22..23] := 0.0;
   Receptura[5].Krok[2].PM[24] := 3101.0;
   Receptura[5].Krok[2].PM[25..30] := 0.0;
   Receptura[5].Krok[3].PM[0] := 0.0;
   Receptura[5].Krok[3].PM[1] := 1.0;
   Receptura[5].Krok[3].PM[2] := 15.0;
   Receptura[5].Krok[3].PM[3] := 10.0;
   Receptura[5].Krok[3].PM[4] := 60.0;
   Receptura[5].Krok[3].PM[5] := 0.5;
   Receptura[5].Krok[3].PM[6] := 600.0;
   Receptura[5].Krok[3].PM[7..9] := 0.0;
   Receptura[5].Krok[3].PM[10] := 40.0;
   Receptura[5].Krok[3].PM[11] := 75.0;
   Receptura[5].Krok[3].PM[12] := 3.0;
   Receptura[5].Krok[3].PM[13] := 70.0;
   Receptura[5].Krok[3].PM[14] := 30.0;
   Receptura[5].Krok[3].PM[15] := 1.0;
   Receptura[5].Krok[3].PM[16] := 10.0;
   Receptura[5].Krok[3].PM[17] := 2.05;
   Receptura[5].Krok[3].PM[18] := 20.0;
   Receptura[5].Krok[3].PM[19] := 300.0;
   Receptura[5].Krok[3].PM[20] := 0.0;
   Receptura[5].Krok[3].PM[21..22] := 1.0;
   Receptura[5].Krok[3].PM[23] := 0.0;
   Receptura[5].Krok[3].PM[24] := 3101.0;
   Receptura[5].Krok[3].PM[25..30] := 0.0;
   Receptura[5].Krok[4].PM[0] := 0.0;
   Receptura[5].Krok[4].PM[1] := 1.0;
   Receptura[5].Krok[4].PM[2] := 15.0;
   Receptura[5].Krok[4].PM[3] := 10.0;
   Receptura[5].Krok[4].PM[4] := 60.0;
   Receptura[5].Krok[4].PM[5] := 0.1;
   Receptura[5].Krok[4].PM[6] := 300.0;
   Receptura[5].Krok[4].PM[7..9] := 0.0;
   Receptura[5].Krok[4].PM[10] := 30.0;
   Receptura[5].Krok[4].PM[11] := 50.0;
   Receptura[5].Krok[4].PM[12] := 3.0;
   Receptura[5].Krok[4].PM[13] := 60.0;
   Receptura[5].Krok[4].PM[14] := 0.0;
   Receptura[5].Krok[4].PM[15] := 1.0;
   Receptura[5].Krok[4].PM[16] := 10.0;
   Receptura[5].Krok[4].PM[17] := 1.75;
   Receptura[5].Krok[4].PM[18] := 20.0;
   Receptura[5].Krok[4].PM[19] := 300.0;
   Receptura[5].Krok[4].PM[20] := 0.0;
   Receptura[5].Krok[4].PM[21..22] := 1.0;
   Receptura[5].Krok[4].PM[23] := 0.0;
   Receptura[5].Krok[4].PM[24] := 3101.0;
   Receptura[5].Krok[4].PM[25..30] := 0.0;
   Receptura[5].Krok[5].PM[0] := 0.0;
   Receptura[5].Krok[5].PM[1] := 1.0;
   Receptura[5].Krok[5].PM[2] := 15.0;
   Receptura[5].Krok[5].PM[3] := 10.0;
   Receptura[5].Krok[5].PM[4] := 60.0;
   Receptura[5].Krok[5].PM[5] := 1.0;
   Receptura[5].Krok[5].PM[6..11] := 0.0;
   Receptura[5].Krok[5].PM[12] := 3.0;
   Receptura[5].Krok[5].PM[13..14] := 0.0;
   Receptura[5].Krok[5].PM[15] := 1.0;
   Receptura[5].Krok[5].PM[16..18] := 0.0;
   Receptura[5].Krok[5].PM[19] := 300.0;
   Receptura[5].Krok[5].PM[20] := 0.0;
   Receptura[5].Krok[5].PM[21] := 1.0;
   Receptura[5].Krok[5].PM[22..23] := 0.0;
   Receptura[5].Krok[5].PM[24] := 3101.0;
   Receptura[5].Krok[5].PM[25..30] := 0.0;
   Receptura[5].Krok[6].PM[0..30] := 0.0;
   Receptura[6].Krok[0].PM[0] := 0.0;
   Receptura[6].Krok[0].PM[1] := 1.0;
   Receptura[6].Krok[0].PM[2] := 18.0;
   Receptura[6].Krok[0].PM[3] := 10.0;
   Receptura[6].Krok[0].PM[4] := 30.0;
   Receptura[6].Krok[0].PM[5] := 1.0;
   Receptura[6].Krok[0].PM[6] := 600.0;
   Receptura[6].Krok[0].PM[7..9] := 0.0;
   Receptura[6].Krok[0].PM[10] := 40.0;
   Receptura[6].Krok[0].PM[11] := 75.0;
   Receptura[6].Krok[0].PM[12] := 3.0;
   Receptura[6].Krok[0].PM[13] := 70.0;
   Receptura[6].Krok[0].PM[14] := 30.0;
   Receptura[6].Krok[0].PM[15] := 1.0;
   Receptura[6].Krok[0].PM[16] := 10.0;
   Receptura[6].Krok[0].PM[17] := 2.05;
   Receptura[6].Krok[0].PM[18] := 20.0;
   Receptura[6].Krok[0].PM[19] := 300.0;
   Receptura[6].Krok[0].PM[20] := 0.0;
   Receptura[6].Krok[0].PM[21..22] := 1.0;
   Receptura[6].Krok[0].PM[23] := 0.0;
   Receptura[6].Krok[0].PM[24] := 9501.0;
   Receptura[6].Krok[0].PM[25..30] := 0.0;
   Receptura[6].Krok[1].PM[0] := 0.0;
   Receptura[6].Krok[1].PM[1] := 1.0;
   Receptura[6].Krok[1].PM[2] := 18.0;
   Receptura[6].Krok[1].PM[3] := 10.0;
   Receptura[6].Krok[1].PM[4] := 30.0;
   Receptura[6].Krok[1].PM[5] := 0.5;
   Receptura[6].Krok[1].PM[6..11] := 0.0;
   Receptura[6].Krok[1].PM[12] := 3.0;
   Receptura[6].Krok[1].PM[13..14] := 0.0;
   Receptura[6].Krok[1].PM[15] := 1.0;
   Receptura[6].Krok[1].PM[16..18] := 0.0;
   Receptura[6].Krok[1].PM[19] := 300.0;
   Receptura[6].Krok[1].PM[20] := 0.0;
   Receptura[6].Krok[1].PM[21] := 1.0;
   Receptura[6].Krok[1].PM[22..23] := 0.0;
   Receptura[6].Krok[1].PM[24] := 9501.0;
   Receptura[6].Krok[1].PM[25..30] := 0.0;
   Receptura[6].Krok[2].PM[0] := 0.0;
   Receptura[6].Krok[2].PM[1] := 1.0;
   Receptura[6].Krok[2].PM[2] := 18.0;
   Receptura[6].Krok[2].PM[3] := 10.0;
   Receptura[6].Krok[2].PM[4] := 30.0;
   Receptura[6].Krok[2].PM[5] := 0.5;
   Receptura[6].Krok[2].PM[6..11] := 0.0;
   Receptura[6].Krok[2].PM[12] := 3.0;
   Receptura[6].Krok[2].PM[13] := 0.0;
   Receptura[6].Krok[2].PM[14] := 30.0;
   Receptura[6].Krok[2].PM[15] := 1.0;
   Receptura[6].Krok[2].PM[16] := 10.0;
   Receptura[6].Krok[2].PM[17..18] := 0.0;
   Receptura[6].Krok[2].PM[19] := 300.0;
   Receptura[6].Krok[2].PM[20] := 0.0;
   Receptura[6].Krok[2].PM[21] := 1.0;
   Receptura[6].Krok[2].PM[22..23] := 0.0;
   Receptura[6].Krok[2].PM[24] := 9501.0;
   Receptura[6].Krok[2].PM[25..30] := 0.0;
   Receptura[6].Krok[3].PM[0] := 0.0;
   Receptura[6].Krok[3].PM[1] := 1.0;
   Receptura[6].Krok[3].PM[2] := 18.0;
   Receptura[6].Krok[3].PM[3] := 10.0;
   Receptura[6].Krok[3].PM[4] := 30.0;
   Receptura[6].Krok[3].PM[5] := 1.0;
   Receptura[6].Krok[3].PM[6] := 600.0;
   Receptura[6].Krok[3].PM[7..9] := 0.0;
   Receptura[6].Krok[3].PM[10] := 40.0;
   Receptura[6].Krok[3].PM[11] := 75.0;
   Receptura[6].Krok[3].PM[12] := 3.0;
   Receptura[6].Krok[3].PM[13] := 70.0;
   Receptura[6].Krok[3].PM[14] := 30.0;
   Receptura[6].Krok[3].PM[15] := 1.0;
   Receptura[6].Krok[3].PM[16] := 10.0;
   Receptura[6].Krok[3].PM[17] := 2.05;
   Receptura[6].Krok[3].PM[18] := 20.0;
   Receptura[6].Krok[3].PM[19] := 300.0;
   Receptura[6].Krok[3].PM[20] := 0.0;
   Receptura[6].Krok[3].PM[21..22] := 1.0;
   Receptura[6].Krok[3].PM[23] := 0.0;
   Receptura[6].Krok[3].PM[24] := 9501.0;
   Receptura[6].Krok[3].PM[25..30] := 0.0;
   Receptura[6].Krok[4].PM[0] := 0.0;
   Receptura[6].Krok[4].PM[1] := 1.0;
   Receptura[6].Krok[4].PM[2] := 18.0;
   Receptura[6].Krok[4].PM[3] := 10.0;
   Receptura[6].Krok[4].PM[4] := 30.0;
   Receptura[6].Krok[4].PM[5] := 0.1;
   Receptura[6].Krok[4].PM[6] := 300.0;
   Receptura[6].Krok[4].PM[7..9] := 0.0;
   Receptura[6].Krok[4].PM[10] := 30.0;
   Receptura[6].Krok[4].PM[11] := 50.0;
   Receptura[6].Krok[4].PM[12] := 3.0;
   Receptura[6].Krok[4].PM[13] := 60.0;
   Receptura[6].Krok[4].PM[14] := 0.0;
   Receptura[6].Krok[4].PM[15] := 1.0;
   Receptura[6].Krok[4].PM[16] := 10.0;
   Receptura[6].Krok[4].PM[17] := 1.75;
   Receptura[6].Krok[4].PM[18] := 20.0;
   Receptura[6].Krok[4].PM[19] := 300.0;
   Receptura[6].Krok[4].PM[20] := 0.0;
   Receptura[6].Krok[4].PM[21..22] := 1.0;
   Receptura[6].Krok[4].PM[23] := 0.0;
   Receptura[6].Krok[4].PM[24] := 9501.0;
   Receptura[6].Krok[4].PM[25..30] := 0.0;
   Receptura[6].Krok[5].PM[0] := 0.0;
   Receptura[6].Krok[5].PM[1] := 1.0;
   Receptura[6].Krok[5].PM[2] := 18.0;
   Receptura[6].Krok[5].PM[3] := 10.0;
   Receptura[6].Krok[5].PM[4] := 30.0;
   Receptura[6].Krok[5].PM[5] := 1.0;
   Receptura[6].Krok[5].PM[6..11] := 0.0;
   Receptura[6].Krok[5].PM[12] := 3.0;
   Receptura[6].Krok[5].PM[13..14] := 0.0;
   Receptura[6].Krok[5].PM[15] := 1.0;
   Receptura[6].Krok[5].PM[16..18] := 0.0;
   Receptura[6].Krok[5].PM[19] := 300.0;
   Receptura[6].Krok[5].PM[20] := 0.0;
   Receptura[6].Krok[5].PM[21] := 1.0;
   Receptura[6].Krok[5].PM[22..23] := 0.0;
   Receptura[6].Krok[5].PM[24] := 9501.0;
   Receptura[6].Krok[5].PM[25..30] := 0.0;
   Receptura[6].Krok[6].PM[0..30] := 0.0;
   Receptura[7].Krok[0].PM[0] := 0.0;
   Receptura[7].Krok[0].PM[1] := 1.0;
   Receptura[7].Krok[0].PM[2] := 17.0;
   Receptura[7].Krok[0].PM[3] := 10.0;
   Receptura[7].Krok[0].PM[4] := 120.0;
   Receptura[7].Krok[0].PM[5] := 1.5;
   Receptura[7].Krok[0].PM[6..11] := 0.0;
   Receptura[7].Krok[0].PM[12] := 3.0;
   Receptura[7].Krok[0].PM[13..14] := 0.0;
   Receptura[7].Krok[0].PM[15] := 1.0;
   Receptura[7].Krok[0].PM[16..18] := 0.0;
   Receptura[7].Krok[0].PM[19] := 300.0;
   Receptura[7].Krok[0].PM[20] := 0.0;
   Receptura[7].Krok[0].PM[21] := 1.0;
   Receptura[7].Krok[0].PM[22] := 0.0;
   Receptura[7].Krok[0].PM[23] := 1.0;
   Receptura[7].Krok[0].PM[24] := 9401.0;
   Receptura[7].Krok[0].PM[25..30] := 0.0;
   Receptura[7].Krok[1].PM[0] := 0.0;
   Receptura[7].Krok[1].PM[1] := 1.0;
   Receptura[7].Krok[1].PM[2] := 17.0;
   Receptura[7].Krok[1].PM[3..4] := 10.0;
   Receptura[7].Krok[1].PM[5] := 1.0;
   Receptura[7].Krok[1].PM[6..11] := 0.0;
   Receptura[7].Krok[1].PM[12] := 3.0;
   Receptura[7].Krok[1].PM[13..14] := 0.0;
   Receptura[7].Krok[1].PM[15] := 1.0;
   Receptura[7].Krok[1].PM[16..18] := 0.0;
   Receptura[7].Krok[1].PM[19] := 300.0;
   Receptura[7].Krok[1].PM[20] := 0.0;
   Receptura[7].Krok[1].PM[21] := 1.0;
   Receptura[7].Krok[1].PM[22] := 0.0;
   Receptura[7].Krok[1].PM[23] := 1.0;
   Receptura[7].Krok[1].PM[24] := 9401.0;
   Receptura[7].Krok[1].PM[25..30] := 0.0;
   Receptura[7].Krok[2].PM[0] := 0.0;
   Receptura[7].Krok[2].PM[1] := 1.0;
   Receptura[7].Krok[2].PM[2] := 17.0;
   Receptura[7].Krok[2].PM[3] := 10.0;
   Receptura[7].Krok[2].PM[4] := 120.0;
   Receptura[7].Krok[2].PM[5] := 0.5;
   Receptura[7].Krok[2].PM[6..11] := 0.0;
   Receptura[7].Krok[2].PM[12] := 3.0;
   Receptura[7].Krok[2].PM[13] := 0.0;
   Receptura[7].Krok[2].PM[14] := 30.0;
   Receptura[7].Krok[2].PM[15] := 1.0;
   Receptura[7].Krok[2].PM[16] := 10.0;
   Receptura[7].Krok[2].PM[17..18] := 0.0;
   Receptura[7].Krok[2].PM[19] := 300.0;
   Receptura[7].Krok[2].PM[20] := 0.0;
   Receptura[7].Krok[2].PM[21] := 1.0;
   Receptura[7].Krok[2].PM[22] := 0.0;
   Receptura[7].Krok[2].PM[23] := 1.0;
   Receptura[7].Krok[2].PM[24] := 9401.0;
   Receptura[7].Krok[2].PM[25..30] := 0.0;
   Receptura[7].Krok[3].PM[0] := 0.0;
   Receptura[7].Krok[3].PM[1] := 1.0;
   Receptura[7].Krok[3].PM[2] := 17.0;
   Receptura[7].Krok[3].PM[3] := 10.0;
   Receptura[7].Krok[3].PM[4] := 120.0;
   Receptura[7].Krok[3].PM[5] := 1.0;
   Receptura[7].Krok[3].PM[6] := 20.0;
   Receptura[7].Krok[3].PM[7..9] := 0.0;
   Receptura[7].Krok[3].PM[10] := 60.0;
   Receptura[7].Krok[3].PM[11] := 75.0;
   Receptura[7].Krok[3].PM[12] := 3.0;
   Receptura[7].Krok[3].PM[13] := 70.0;
   Receptura[7].Krok[3].PM[14] := 30.0;
   Receptura[7].Krok[3].PM[15] := 1.0;
   Receptura[7].Krok[3].PM[16] := 10.0;
   Receptura[7].Krok[3].PM[17] := 2.05;
   Receptura[7].Krok[3].PM[18] := 20.0;
   Receptura[7].Krok[3].PM[19] := 300.0;
   Receptura[7].Krok[3].PM[20..21] := 0.0;
   Receptura[7].Krok[3].PM[22..23] := 1.0;
   Receptura[7].Krok[3].PM[24] := 9401.0;
   Receptura[7].Krok[3].PM[25..30] := 0.0;
   Receptura[7].Krok[4].PM[0] := 0.0;
   Receptura[7].Krok[4].PM[1] := 1.0;
   Receptura[7].Krok[4].PM[2] := 17.0;
   Receptura[7].Krok[4].PM[3] := 10.0;
   Receptura[7].Krok[4].PM[4] := 120.0;
   Receptura[7].Krok[4].PM[5] := 0.1;
   Receptura[7].Krok[4].PM[6] := 10.0;
   Receptura[7].Krok[4].PM[7..9] := 0.0;
   Receptura[7].Krok[4].PM[10] := 35.0;
   Receptura[7].Krok[4].PM[11] := 50.0;
   Receptura[7].Krok[4].PM[12] := 3.0;
   Receptura[7].Krok[4].PM[13] := 60.0;
   Receptura[7].Krok[4].PM[14] := 0.0;
   Receptura[7].Krok[4].PM[15] := 1.0;
   Receptura[7].Krok[4].PM[16] := 10.0;
   Receptura[7].Krok[4].PM[17] := 1.75;
   Receptura[7].Krok[4].PM[18] := 20.0;
   Receptura[7].Krok[4].PM[19] := 300.0;
   Receptura[7].Krok[4].PM[20..21] := 0.0;
   Receptura[7].Krok[4].PM[22..23] := 1.0;
   Receptura[7].Krok[4].PM[24] := 9401.0;
   Receptura[7].Krok[4].PM[25..30] := 0.0;
   Receptura[7].Krok[5].PM[0] := 0.0;
   Receptura[7].Krok[5].PM[1] := 1.0;
   Receptura[7].Krok[5].PM[2] := 17.0;
   Receptura[7].Krok[5].PM[3] := 10.0;
   Receptura[7].Krok[5].PM[4] := 120.0;
   Receptura[7].Krok[5].PM[5] := 1.5;
   Receptura[7].Krok[5].PM[6..11] := 0.0;
   Receptura[7].Krok[5].PM[12] := 3.0;
   Receptura[7].Krok[5].PM[13..14] := 0.0;
   Receptura[7].Krok[5].PM[15] := 1.0;
   Receptura[7].Krok[5].PM[16..18] := 0.0;
   Receptura[7].Krok[5].PM[19] := 300.0;
   Receptura[7].Krok[5].PM[20] := 0.0;
   Receptura[7].Krok[5].PM[21] := 1.0;
   Receptura[7].Krok[5].PM[22] := 0.0;
   Receptura[7].Krok[5].PM[23] := 1.0;
   Receptura[7].Krok[5].PM[24] := 9401.0;
   Receptura[7].Krok[5].PM[25..30] := 0.0;
   Receptura[7].Krok[6].PM[0..30] := 0.0;
   Receptura[8].Krok[0].PM[0] := 0.0;
   Receptura[8].Krok[0].PM[1] := 1.0;
   Receptura[8].Krok[0].PM[2] := 25.0;
   Receptura[8].Krok[0].PM[3] := 10.0;
   Receptura[8].Krok[0].PM[4] := 120.0;
   Receptura[8].Krok[0].PM[5] := 0.5;
   Receptura[8].Krok[0].PM[6..11] := 0.0;
   Receptura[8].Krok[0].PM[12] := 3.0;
   Receptura[8].Krok[0].PM[13] := 0.0;
   Receptura[8].Krok[0].PM[14] := 30.0;
   Receptura[8].Krok[0].PM[15] := 1.0;
   Receptura[8].Krok[0].PM[16] := 10.0;
   Receptura[8].Krok[0].PM[17..18] := 0.0;
   Receptura[8].Krok[0].PM[19] := 300.0;
   Receptura[8].Krok[0].PM[20..23] := 0.0;
   Receptura[8].Krok[0].PM[24] := 9401.0;
   Receptura[8].Krok[0].PM[25..30] := 0.0;
   Receptura[8].Krok[1].PM[0] := 0.0;
   Receptura[8].Krok[1].PM[1] := 1.0;
   Receptura[8].Krok[1].PM[2] := 25.0;
   Receptura[8].Krok[1].PM[3] := 10.0;
   Receptura[8].Krok[1].PM[4] := 120.0;
   Receptura[8].Krok[1].PM[5] := 1.0;
   Receptura[8].Krok[1].PM[6..11] := 0.0;
   Receptura[8].Krok[1].PM[12] := 3.0;
   Receptura[8].Krok[1].PM[13..14] := 0.0;
   Receptura[8].Krok[1].PM[15] := 1.0;
   Receptura[8].Krok[1].PM[16..18] := 0.0;
   Receptura[8].Krok[1].PM[19] := 300.0;
   Receptura[8].Krok[1].PM[20..23] := 0.0;
   Receptura[8].Krok[1].PM[24] := 9401.0;
   Receptura[8].Krok[1].PM[25..30] := 0.0;
   Receptura[8].Krok[2].PM[0] := 0.0;
   Receptura[8].Krok[2].PM[1] := 1.0;
   Receptura[8].Krok[2].PM[2] := 25.0;
   Receptura[8].Krok[2].PM[3] := 10.0;
   Receptura[8].Krok[2].PM[4] := 120.0;
   Receptura[8].Krok[2].PM[5] := 0.5;
   Receptura[8].Krok[2].PM[6..11] := 0.0;
   Receptura[8].Krok[2].PM[12] := 3.0;
   Receptura[8].Krok[2].PM[13] := 0.0;
   Receptura[8].Krok[2].PM[14] := 30.0;
   Receptura[8].Krok[2].PM[15] := 1.0;
   Receptura[8].Krok[2].PM[16] := 10.0;
   Receptura[8].Krok[2].PM[17..18] := 0.0;
   Receptura[8].Krok[2].PM[19] := 300.0;
   Receptura[8].Krok[2].PM[20..23] := 0.0;
   Receptura[8].Krok[2].PM[24] := 9401.0;
   Receptura[8].Krok[2].PM[25..30] := 0.0;
   Receptura[8].Krok[3].PM[0] := 0.0;
   Receptura[8].Krok[3].PM[1] := 1.0;
   Receptura[8].Krok[3].PM[2] := 25.0;
   Receptura[8].Krok[3].PM[3] := 10.0;
   Receptura[8].Krok[3].PM[4] := 120.0;
   Receptura[8].Krok[3].PM[5] := 1.0;
   Receptura[8].Krok[3].PM[6] := 900.0;
   Receptura[8].Krok[3].PM[7..9] := 0.0;
   Receptura[8].Krok[3].PM[10] := 60.0;
   Receptura[8].Krok[3].PM[11] := 75.0;
   Receptura[8].Krok[3].PM[12] := 3.0;
   Receptura[8].Krok[3].PM[13] := 70.0;
   Receptura[8].Krok[3].PM[14] := 30.0;
   Receptura[8].Krok[3].PM[15] := 1.0;
   Receptura[8].Krok[3].PM[16] := 10.0;
   Receptura[8].Krok[3].PM[17] := 2.05;
   Receptura[8].Krok[3].PM[18] := 20.0;
   Receptura[8].Krok[3].PM[19] := 300.0;
   Receptura[8].Krok[3].PM[20..21] := 0.0;
   Receptura[8].Krok[3].PM[22] := 1.0;
   Receptura[8].Krok[3].PM[23] := 0.0;
   Receptura[8].Krok[3].PM[24] := 9401.0;
   Receptura[8].Krok[3].PM[25..30] := 0.0;
   Receptura[8].Krok[4].PM[0] := 0.0;
   Receptura[8].Krok[4].PM[1] := 1.0;
   Receptura[8].Krok[4].PM[2] := 25.0;
   Receptura[8].Krok[4].PM[3] := 10.0;
   Receptura[8].Krok[4].PM[4] := 120.0;
   Receptura[8].Krok[4].PM[5] := 0.1;
   Receptura[8].Krok[4].PM[6] := 300.0;
   Receptura[8].Krok[4].PM[7..9] := 0.0;
   Receptura[8].Krok[4].PM[10] := 35.0;
   Receptura[8].Krok[4].PM[11] := 50.0;
   Receptura[8].Krok[4].PM[12] := 3.0;
   Receptura[8].Krok[4].PM[13] := 60.0;
   Receptura[8].Krok[4].PM[14] := 0.0;
   Receptura[8].Krok[4].PM[15] := 1.0;
   Receptura[8].Krok[4].PM[16] := 10.0;
   Receptura[8].Krok[4].PM[17] := 1.75;
   Receptura[8].Krok[4].PM[18] := 20.0;
   Receptura[8].Krok[4].PM[19] := 300.0;
   Receptura[8].Krok[4].PM[20..21] := 0.0;
   Receptura[8].Krok[4].PM[22] := 1.0;
   Receptura[8].Krok[4].PM[23] := 0.0;
   Receptura[8].Krok[4].PM[24] := 9401.0;
   Receptura[8].Krok[4].PM[25..30] := 0.0;
   Receptura[8].Krok[5].PM[0] := 0.0;
   Receptura[8].Krok[5].PM[1] := 1.0;
   Receptura[8].Krok[5].PM[2] := 25.0;
   Receptura[8].Krok[5].PM[3] := 10.0;
   Receptura[8].Krok[5].PM[4] := 120.0;
   Receptura[8].Krok[5].PM[5] := 1.5;
   Receptura[8].Krok[5].PM[6..11] := 0.0;
   Receptura[8].Krok[5].PM[12] := 3.0;
   Receptura[8].Krok[5].PM[13..14] := 0.0;
   Receptura[8].Krok[5].PM[15] := 1.0;
   Receptura[8].Krok[5].PM[16..18] := 0.0;
   Receptura[8].Krok[5].PM[19] := 300.0;
   Receptura[8].Krok[5].PM[20..23] := 0.0;
   Receptura[8].Krok[5].PM[24] := 9401.0;
   Receptura[8].Krok[5].PM[25..30] := 0.0;
   Receptura[8].Krok[6].PM[0..30] := 0.0;
   Receptura[9].Krok[0].PM[0..30] := 0.0;
   Receptura[9].Krok[1].PM[0..30] := 0.0;
   Receptura[9].Krok[2].PM[0..30] := 0.0;
   Receptura[9].Krok[3].PM[0..30] := 0.0;
   Receptura[9].Krok[4].PM[0..30] := 0.0;
   Receptura[9].Krok[5].PM[0..30] := 0.0;
   Receptura[9].Krok[6].PM[0..30] := 0.0;
   Receptura[10].Krok[0].PM[0..30] := 0.0;
   Receptura[10].Krok[1].PM[0..30] := 0.0;
   Receptura[10].Krok[2].PM[0..30] := 0.0;
   Receptura[10].Krok[3].PM[0..30] := 0.0;
   Receptura[10].Krok[4].PM[0..30] := 0.0;
   Receptura[10].Krok[5].PM[0..30] := 0.0;
   Receptura[10].Krok[6].PM[0..30] := 0.0;
   Receptura[11].Krok[0].PM[0..30] := 0.0;
   Receptura[11].Krok[1].PM[0..30] := 0.0;
   Receptura[11].Krok[2].PM[0..30] := 0.0;
   Receptura[11].Krok[3].PM[0..30] := 0.0;
   Receptura[11].Krok[4].PM[0..30] := 0.0;
   Receptura[11].Krok[5].PM[0..30] := 0.0;
   Receptura[11].Krok[6].PM[0..30] := 0.0;
   Receptura[12].Krok[0].PM[0..30] := 0.0;
   Receptura[12].Krok[1].PM[0..30] := 0.0;
   Receptura[12].Krok[2].PM[0..30] := 0.0;
   Receptura[12].Krok[3].PM[0..30] := 0.0;
   Receptura[12].Krok[4].PM[0..30] := 0.0;
   Receptura[12].Krok[5].PM[0..30] := 0.0;
   Receptura[12].Krok[6].PM[0..30] := 0.0;
   Receptura[13].Krok[0].PM[0..30] := 0.0;
   Receptura[13].Krok[1].PM[0..30] := 0.0;
   Receptura[13].Krok[2].PM[0..30] := 0.0;
   Receptura[13].Krok[3].PM[0..30] := 0.0;
   Receptura[13].Krok[4].PM[0..30] := 0.0;
   Receptura[13].Krok[5].PM[0..30] := 0.0;
   Receptura[13].Krok[6].PM[0..30] := 0.0;
   Receptura[14].Krok[0].PM[0..30] := 0.0;
   Receptura[14].Krok[1].PM[0..30] := 0.0;
   Receptura[14].Krok[2].PM[0..30] := 0.0;
   Receptura[14].Krok[3].PM[0..30] := 0.0;
   Receptura[14].Krok[4].PM[0..30] := 0.0;
   Receptura[14].Krok[5].PM[0..30] := 0.0;
   Receptura[14].Krok[6].PM[0..30] := 0.0;
   Receptura[15].Krok[0].PM[0..30] := 0.0;
   Receptura[15].Krok[1].PM[0..30] := 0.0;
   Receptura[15].Krok[2].PM[0..30] := 0.0;
   Receptura[15].Krok[3].PM[0..30] := 0.0;
   Receptura[15].Krok[4].PM[0..30] := 0.0;
   Receptura[15].Krok[5].PM[0..30] := 0.0;
   Receptura[15].Krok[6].PM[0..30] := 0.0;
   Receptura[16].Krok[0].PM[0..30] := 0.0;
   Receptura[16].Krok[1].PM[0..30] := 0.0;
   Receptura[16].Krok[2].PM[0..30] := 0.0;
   Receptura[16].Krok[3].PM[0..30] := 0.0;
   Receptura[16].Krok[4].PM[0..30] := 0.0;
   Receptura[16].Krok[5].PM[0..30] := 0.0;
   Receptura[16].Krok[6].PM[0..30] := 0.0;
   Receptura[17].Krok[0].PM[0..30] := 0.0;
   Receptura[17].Krok[1].PM[0..30] := 0.0;
   Receptura[17].Krok[2].PM[0..30] := 0.0;
   Receptura[17].Krok[3].PM[0..30] := 0.0;
   Receptura[17].Krok[4].PM[0..30] := 0.0;
   Receptura[17].Krok[5].PM[0..30] := 0.0;
   Receptura[17].Krok[6].PM[0..30] := 0.0;
   Receptura[18].Krok[0].PM[0..30] := 0.0;
   Receptura[18].Krok[1].PM[0..30] := 0.0;
   Receptura[18].Krok[2].PM[0..30] := 0.0;
   Receptura[18].Krok[3].PM[0..30] := 0.0;
   Receptura[18].Krok[4].PM[0..30] := 0.0;
   Receptura[18].Krok[5].PM[0..30] := 0.0;
   Receptura[18].Krok[6].PM[0..30] := 0.0;
   Receptura[19].Krok[0].PM[0..30] := 0.0;
   Receptura[19].Krok[1].PM[0..30] := 0.0;
   Receptura[19].Krok[2].PM[0..30] := 0.0;
   Receptura[19].Krok[3].PM[0..30] := 0.0;
   Receptura[19].Krok[4].PM[0..30] := 0.0;
   Receptura[19].Krok[5].PM[0..30] := 0.0;
   Receptura[19].Krok[6].PM[0..30] := 0.0;
   Receptura[20].Krok[0].PM[0] := 0.0;
   Receptura[20].Krok[0].PM[1] := 1.0;
   Receptura[20].Krok[0].PM[2] := 25.0;
   Receptura[20].Krok[0].PM[3] := 10.0;
   Receptura[20].Krok[0].PM[4] := 120.0;
   Receptura[20].Krok[0].PM[5] := 1.0;
   Receptura[20].Krok[0].PM[6..11] := 0.0;
   Receptura[20].Krok[0].PM[12] := 3.0;
   Receptura[20].Krok[0].PM[13..14] := 0.0;
   Receptura[20].Krok[0].PM[15] := 1.0;
   Receptura[20].Krok[0].PM[16..18] := 0.0;
   Receptura[20].Krok[0].PM[19] := 300.0;
   Receptura[20].Krok[0].PM[20..23] := 0.0;
   Receptura[20].Krok[0].PM[24] := 9401.0;
   Receptura[20].Krok[0].PM[25..30] := 0.0;
   Receptura[20].Krok[1].PM[0] := 0.0;
   Receptura[20].Krok[1].PM[1] := 1.0;
   Receptura[20].Krok[1].PM[2] := 25.0;
   Receptura[20].Krok[1].PM[3] := 10.0;
   Receptura[20].Krok[1].PM[4] := 120.0;
   Receptura[20].Krok[1].PM[5] := 1.0;
   Receptura[20].Krok[1].PM[6..11] := 0.0;
   Receptura[20].Krok[1].PM[12] := 3.0;
   Receptura[20].Krok[1].PM[13..14] := 0.0;
   Receptura[20].Krok[1].PM[15] := 1.0;
   Receptura[20].Krok[1].PM[16..18] := 0.0;
   Receptura[20].Krok[1].PM[19] := 300.0;
   Receptura[20].Krok[1].PM[20..23] := 0.0;
   Receptura[20].Krok[1].PM[24] := 9401.0;
   Receptura[20].Krok[1].PM[25..30] := 0.0;
   Receptura[20].Krok[2].PM[0] := 0.0;
   Receptura[20].Krok[2].PM[1] := 1.0;
   Receptura[20].Krok[2].PM[2] := 25.0;
   Receptura[20].Krok[2].PM[3] := 10.0;
   Receptura[20].Krok[2].PM[4] := 120.0;
   Receptura[20].Krok[2].PM[5] := 0.5;
   Receptura[20].Krok[2].PM[6..11] := 0.0;
   Receptura[20].Krok[2].PM[12] := 3.0;
   Receptura[20].Krok[2].PM[13] := 0.0;
   Receptura[20].Krok[2].PM[14] := 30.0;
   Receptura[20].Krok[2].PM[15] := 1.0;
   Receptura[20].Krok[2].PM[16] := 10.0;
   Receptura[20].Krok[2].PM[17..18] := 0.0;
   Receptura[20].Krok[2].PM[19] := 300.0;
   Receptura[20].Krok[2].PM[20..23] := 0.0;
   Receptura[20].Krok[2].PM[24] := 9401.0;
   Receptura[20].Krok[2].PM[25..30] := 0.0;
   Receptura[20].Krok[3].PM[0] := 0.0;
   Receptura[20].Krok[3].PM[1] := 1.0;
   Receptura[20].Krok[3].PM[2] := 25.0;
   Receptura[20].Krok[3].PM[3] := 10.0;
   Receptura[20].Krok[3].PM[4] := 120.0;
   Receptura[20].Krok[3].PM[5] := 1.0;
   Receptura[20].Krok[3].PM[6] := 900.0;
   Receptura[20].Krok[3].PM[7..9] := 0.0;
   Receptura[20].Krok[3].PM[10] := 60.0;
   Receptura[20].Krok[3].PM[11] := 75.0;
   Receptura[20].Krok[3].PM[12] := 3.0;
   Receptura[20].Krok[3].PM[13] := 70.0;
   Receptura[20].Krok[3].PM[14] := 30.0;
   Receptura[20].Krok[3].PM[15] := 1.0;
   Receptura[20].Krok[3].PM[16] := 10.0;
   Receptura[20].Krok[3].PM[17] := 2.05;
   Receptura[20].Krok[3].PM[18] := 20.0;
   Receptura[20].Krok[3].PM[19] := 300.0;
   Receptura[20].Krok[3].PM[20..21] := 0.0;
   Receptura[20].Krok[3].PM[22] := 1.0;
   Receptura[20].Krok[3].PM[23] := 0.0;
   Receptura[20].Krok[3].PM[24] := 9401.0;
   Receptura[20].Krok[3].PM[25..30] := 0.0;
   Receptura[20].Krok[4].PM[0] := 0.0;
   Receptura[20].Krok[4].PM[1] := 1.0;
   Receptura[20].Krok[4].PM[2] := 25.0;
   Receptura[20].Krok[4].PM[3] := 10.0;
   Receptura[20].Krok[4].PM[4] := 120.0;
   Receptura[20].Krok[4].PM[5] := 0.1;
   Receptura[20].Krok[4].PM[6] := 300.0;
   Receptura[20].Krok[4].PM[7..9] := 0.0;
   Receptura[20].Krok[4].PM[10] := 35.0;
   Receptura[20].Krok[4].PM[11] := 50.0;
   Receptura[20].Krok[4].PM[12] := 3.0;
   Receptura[20].Krok[4].PM[13] := 60.0;
   Receptura[20].Krok[4].PM[14] := 0.0;
   Receptura[20].Krok[4].PM[15] := 1.0;
   Receptura[20].Krok[4].PM[16] := 10.0;
   Receptura[20].Krok[4].PM[17] := 1.75;
   Receptura[20].Krok[4].PM[18] := 20.0;
   Receptura[20].Krok[4].PM[19] := 300.0;
   Receptura[20].Krok[4].PM[20..21] := 0.0;
   Receptura[20].Krok[4].PM[22] := 1.0;
   Receptura[20].Krok[4].PM[23] := 0.0;
   Receptura[20].Krok[4].PM[24] := 9401.0;
   Receptura[20].Krok[4].PM[25..30] := 0.0;
   Receptura[20].Krok[5].PM[0] := 0.0;
   Receptura[20].Krok[5].PM[1] := 1.0;
   Receptura[20].Krok[5].PM[2] := 25.0;
   Receptura[20].Krok[5].PM[3] := 10.0;
   Receptura[20].Krok[5].PM[4] := 120.0;
   Receptura[20].Krok[5].PM[5] := 1.5;
   Receptura[20].Krok[5].PM[6..11] := 0.0;
   Receptura[20].Krok[5].PM[12] := 3.0;
   Receptura[20].Krok[5].PM[13..14] := 0.0;
   Receptura[20].Krok[5].PM[15] := 1.0;
   Receptura[20].Krok[5].PM[16..18] := 0.0;
   Receptura[20].Krok[5].PM[19] := 300.0;
   Receptura[20].Krok[5].PM[20..23] := 0.0;
   Receptura[20].Krok[5].PM[24] := 9401.0;
   Receptura[20].Krok[5].PM[25..30] := 0.0;
   Receptura[20].Krok[6].PM[0..30] := 0.0;
   "receptura-1".CLK := FALSE;
   "receptura-1".Q := FALSE;
   "receptura-1".Stat_Bit := FALSE;
   "receptura+1".CLK := FALSE;
   "receptura+1".Q := FALSE;
   "receptura+1".Stat_Bit := FALSE;
   wybór_recept.CLK := FALSE;
   wybór_recept.Q := FALSE;
   wybór_recept.Stat_Bit := FALSE;
   kopiuj.CLK := FALSE;
   kopiuj.Q := FALSE;
   kopiuj.Stat_Bit := FALSE;
   wklej.CLK := FALSE;
   wklej.Q := FALSE;
   wklej.Stat_Bit := FALSE;
   zapisz.CLK := FALSE;
   zapisz.Q := FALSE;
   zapisz.Stat_Bit := FALSE;
   użyj.CLK := FALSE;
   użyj.Q := FALSE;
   użyj.Stat_Bit := FALSE;
   "krok+".CLK := FALSE;
   "krok+".Q := FALSE;
   "krok+".Stat_Bit := FALSE;
   "krok-".CLK := FALSE;
   "krok-".Q := FALSE;
   "krok-".Stat_Bit := FALSE;
   wybór_kroku.CLK := FALSE;
   wybór_kroku.Q := FALSE;
   wybór_kroku.Stat_Bit := FALSE;
END_DATA_BLOCK

DATA_BLOCK "Tor2_alarmy"   // DB11
{ DB_Accessible_From_OPC_UA := 'FALSE' }
VERSION : 0.1
// stored: AutoNumber true, DBAccessibleFromOPCUA false, InstanceOfName FB_obsluga_alarmow, InstanceOfType FB
"FB_obsluga_alarmow"
BEGIN
END_DATA_BLOCK
